// TIA Portal project "PID_NIVEL_TANQUE" (V19)

(* hardware
DEVICE "S7-1200 station_1"  S7-1200 Station
   slot 0: "Rack_0"  S7-1200 Rack  Rack  V1.0
   slot 1: "PID_NIVEL_TANQUE"  CPU 1214C DC/DC/Rly  6ES7 214-1HG40-0XB0  V4.6
   slot 2: "AI 4x13BIT/AQ 2x14BIT_1"  6ES7 234-4HE32-0XB0  V2.1
*)

// ===== PLC "PID_NIVEL_TANQUE"  CPU 1214C DC/DC/Rly =====

VAR_GLOBAL   // PLC tag table "Default tag table"
   "I_Liga" AT %I0.0 : Bool;
   "Q_Sys_Hablitado" AT %Q0.0 : Bool;
   "I_Desliga" AT %I0.1 : Bool;
   "sensor_unormalized" AT %IW96 : Int;
   "sensor_normalized" AT %MD0 : Real;
   "sensor_scaled" AT %MD4 : Real;
   "sp" AT %MW8 : Int;
   "pot_bomba" AT %QD2 : Real;
   "pot_bomba_norm" AT %MD10 : Real;
   "pot_bomba_scaled" AT %MW14 : Int;
   "out_velocidade_bomba" AT %QW96 : Int;
END_VAR

ORGANIZATION_BLOCK "Main"   // OB1, LAD, ProgramCycle
TITLE = "Main Program Sweep (Cycle)"
{ S7_Optimized_Access := 'TRUE' }
VERSION : 0.1
   VAR_INPUT
      Initial_Call : Bool;   // Initial call of this OB
      Remanence : Bool;   // =True, if remanent data are available
   END_VAR
BEGIN

REGION Network 1
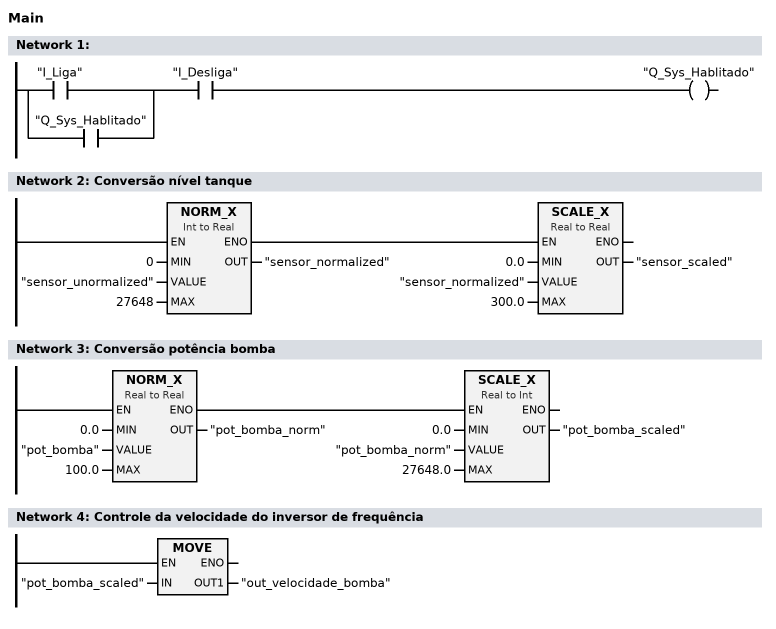
   RUNG wire#powerrail
      Contact( "I_Liga" )
      wire#w1
      Contact( "I_Desliga" )
      Coil( "Q_Sys_Hablitado" )
   END_RUNG
   RUNG wire#powerrail
      Contact( "Q_Sys_Hablitado" )
   END_RUNG wire#w1
   // the same network as SCL:
   "Q_Sys_Hablitado" := ("I_Liga" OR "Q_Sys_Hablitado") AND "I_Desliga";
END_REGION

REGION Network 2: Conversão nível tanque
   RUNG wire#powerrail
      { S7_Templates := "[SrcType := Int, DestType := Real]" } Normalize(min := 0, value := "sensor_unormalized", max := 27648, out => "sensor_normalized")
      { S7_Templates := "[SrcType := Real, DestType := Real]" } Scale(min := 0.0, value := "sensor_normalized", max := 300.0, out => "sensor_scaled")
   END_RUNG
   // the same network as SCL:
   "sensor_normalized" := NORM_X(MIN := 0, VALUE := "sensor_unormalized", MAX := 27648);
   "sensor_scaled" := SCALE_X(MIN := 0.0, VALUE := "sensor_normalized", MAX := 300.0);
END_REGION

REGION Network 3: Conversão potência bomba
   RUNG wire#powerrail
      { S7_Templates := "[SrcType := Real, DestType := Real]" } Normalize(min := 0.0, value := "pot_bomba", max := 100.0, out => "pot_bomba_norm")
      { S7_Templates := "[SrcType := Real, DestType := Int]" } Scale(min := 0.0, value := "pot_bomba_norm", max := 27648.0, out => "pot_bomba_scaled")
   END_RUNG
   // the same network as SCL:
   "pot_bomba_norm" := NORM_X(MIN := 0.0, VALUE := "pot_bomba", MAX := 100.0);
   "pot_bomba_scaled" := SCALE_X(MIN := 0.0, VALUE := "pot_bomba_norm", MAX := 27648.0);
END_REGION

REGION Network 4: Controle da velocidade do inversor de frequência
   RUNG wire#powerrail
      Move(in := "pot_bomba_scaled", out1 => "out_velocidade_bomba")
   END_RUNG
   // the same network as SCL:
   "out_velocidade_bomba" := "pot_bomba_scaled";
END_REGION
END_ORGANIZATION_BLOCK

ORGANIZATION_BLOCK "CyclicInterrupt"   // OB30, LAD, CyclicInterrupt
{ S7_Optimized_Access := 'TRUE' }
VERSION : 0.1
   VAR_INPUT
      Initial_Call : Bool;   // Initial call of this OB
      Event_Count : Int;   // Events discarded
   END_VAR
BEGIN

REGION Network 1: PID - Organization Block
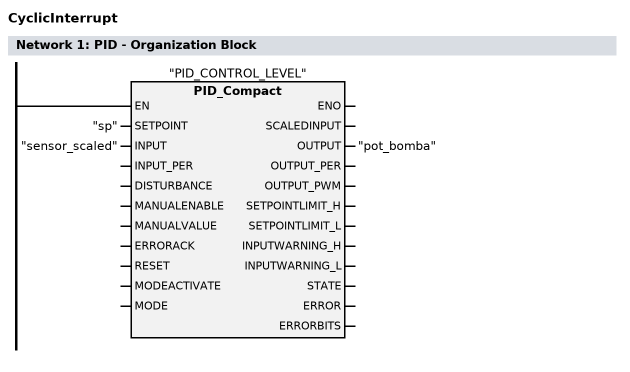
   "PID_CONTROL_LEVEL"(Setpoint := "sp", Input := "sensor_scaled", Output => "pot_bomba");   // PID_Compact
END_REGION
END_ORGANIZATION_BLOCK